SUBAPPLICATION Uebung_160 (* Motor Links/Rechtslauf *)
  (* Standard: 61499-2; Description: Copyright (c) 2023 Meisterschulen am Ostbahnhof This program and the accompanying materials are made available under the terms of the Eclipse Public License 2.0 which is available at https://www.eclipse.org/legal/epl-2.0/ SPDX-License-Identifier: EPL-2.0 *)
  (* Version 1.0, 2023-10-23, Franz Höpfinger, Meisterschulen am Ostbahnhof, initial API and implementation and/or initial documentation *)
  PACKAGE Uebungen;
  IMPORT logiBUS::io::DI::logiBUS_DI::Input_I1;
  IMPORT logiBUS::io::DI::logiBUS_DI::Input_I2;
  IMPORT logiBUS::io::DQ::logiBUS_DO::Output_Q5;
  IMPORT logiBUS::io::DQ::logiBUS_DO::Output_Q56;
  IMPORT logiBUS::io::DQ::logiBUS_DO::Output_Q6;
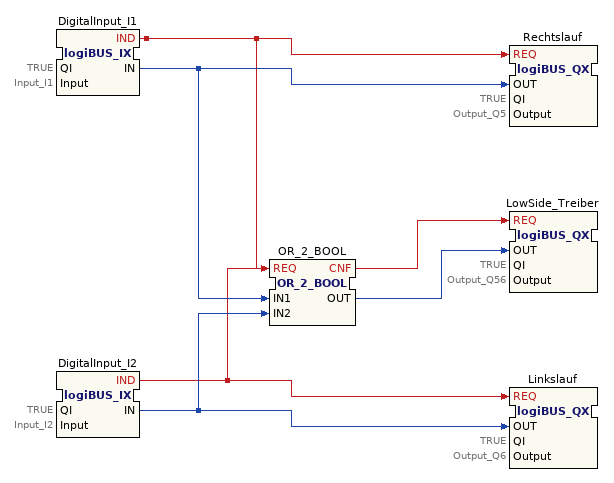
  FBS
    Linkslauf : logiBUS::io::DQ::logiBUS_QX(QI := TRUE, Output := Output_Q6);
    DigitalInput_I2 : logiBUS::io::DI::logiBUS_IX(QI := TRUE, Input := Input_I2);
    OR_2_BOOL : iec61131::booleanOperators::OR_2_BOOL;
    DigitalInput_I1 : logiBUS::io::DI::logiBUS_IX(QI := TRUE, Input := Input_I1);
    Rechtslauf : logiBUS::io::DQ::logiBUS_QX(QI := TRUE, Output := Output_Q5);
    LowSide_Treiber : logiBUS::io::DQ::logiBUS_QX(QI := TRUE, Output := Output_Q56);
  END_FBS
  EVENT_CONNECTIONS
    DigitalInput_I2.IND TO Linkslauf.REQ;
    DigitalInput_I1.IND TO Rechtslauf.REQ;
    OR_2_BOOL.CNF TO LowSide_Treiber.REQ;
    DigitalInput_I2.IND TO OR_2_BOOL.REQ;
    DigitalInput_I1.IND TO OR_2_BOOL.REQ;
  END_CONNECTIONS
  DATA_CONNECTIONS
    DigitalInput_I2.IN TO Linkslauf.OUT;
    DigitalInput_I1.IN TO Rechtslauf.OUT;
    OR_2_BOOL.OUT TO LowSide_Treiber.OUT;
    DigitalInput_I1.IN TO OR_2_BOOL.IN1;
    DigitalInput_I2.IN TO OR_2_BOOL.IN2;
  END_CONNECTIONS
END_SUBAPPLICATION
